TYPE ST_IndexedPositionLinks :
	STRUCT
		Front				: REFERENCE TO ST_DirectionalControls;
		Rear				: REFERENCE TO ST_DirectionalControls;
		Left				: REFERENCE TO ST_DirectionalControls;
		Right				: REFERENCE TO ST_DirectionalControls;
	END_STRUCT
END_TYPE

(* stored: Version 1.1.0.1, ProductVersion 3.1.4024.12
   DUT ST_IndexedPositionLinks: Id {e30ffb78-c0b7-406f-978a-b16632593a4c} *)
